FUNCTION proj5_TupleStruct_1: LREAL
{ S7_Optimized_Access := 'true' }
    VAR_INPUT
        tuple: TupleStruct_1;
    END_VAR

BEGIN
    proj5_TupleStruct_1 := tuple.field5;
END_FUNCTION
